TYPE T_PACK_Barcode : STRING(cMAX_PACKCODE_LENGHT);
END_TYPE

(* stored: Version 1.1.0.1
   DUT T_PACK_Barcode: Id {3fb78c0e-b306-4ef9-a22e-aa7b80fb5f54} *)
